FUNCTION Convert_REAL_TO_DINT : Hresult
VAR_INPUT
	in : REAL;
	out : REFERENCE TO DINT;
END_VAR
VAR
	converted : DINT;
END_VAR
VAR CONSTANT
	INCOMPATIBLE : HRESULT := 16#9811070E;
END_VAR

converted := REAL_TO_DINT(in);

IF (DINT_TO_REAL(converted) <> in) THEN
	Convert_REAL_TO_DINT := INCOMPATIBLE;
	RETURN;
END_IF

out := converted;

END_FUNCTION

(* stored: Version 1.1.0.1, ProductVersion 3.1.4024.12
   POU Convert_REAL_TO_DINT: Id {138cc396-7d89-4639-8cb4-d8f068bb9068}, SpecialFunc None *)
